INTERFACE I_GantryConfigProvider

PROPERTY Config : ST_GantryXYZ_Config
GET
END_GET
SET
END_SET
END_PROPERTY

END_INTERFACE

(* stored: Version 1.1.0.1, ProductVersion 3.1.4024.15
   Itf I_GantryConfigProvider: Id {9e9211f9-23d5-4d2e-9d8e-11348c2e2fe3}
   Property Config: Id {b6f02373-2c30-467f-8952-0a308543758d}
   Get Get: Id {4e10ac90-300e-4568-8d68-214ce6fdfbbc}
   Set Set: Id {caa34027-0b92-4790-8608-e089381308d6} *)
